(* PLC project RLY08, INSA Strasbourg RLY08 1.0, author Mathieu Giamberini *)
(* stored: creationDateTime 2024-11-13T08:40:00, modificationDateTime 2024-10-04T15:56:57 *)

TYPE RLY08 : STRUCT
  CurrentAdress : BYTE := 16#00;
  WantAddress : BYTE := 16#00;
END_STRUCT;
END_TYPE

(* Set the state of the specified relay on the specifeid RLY08 board *)
FUNCTION_BLOCK RLY_1
  VAR_INPUT
    B_AD : BYTE;  (* Board I2C Address *)
    P_AD : BYTE;  (* Pin Address *)
    RLY : BOOL;  (* Pin state *)
  END_VAR

            
          
END_FUNCTION_BLOCK

(* Set the states relays on the specified RLY08 board *)
FUNCTION_BLOCK RLY_8
  VAR_INPUT
    B_AD : BYTE;  (* Board I2C Address *)
    RLY1 : BOOL;  (* Pin state *)
    RLY2 : BOOL;  (* Pin x_0 state *)
    RLY3 : BOOL;  (* Pin x_1 state *)
    RLY4 : BOOL;  (* Pin x_2 state *)
    RLY5 : BOOL;  (* Pin x_3 state *)
    RLY6 : BOOL;  (* Pin x_4 state *)
    RLY7 : BOOL;  (* Pin x_5 state *)
    RLY8 : BOOL;  (* Pin x_6 state *)
  END_VAR

            
          
END_FUNCTION_BLOCK

(* Set the board address to the wanted one and update the config *)
FUNCTION_BLOCK SET_ADDR
  VAR_INPUT
    CONFIG : BYTE;  (* Board Config *)
  END_VAR
  VAR_OUTPUT
    CONFIG : BYTE;  (* Board Config *)
  END_VAR

            
          
END_FUNCTION_BLOCK
